{attribute 'linkalways'} 
{attribute 'no_explicit_call' := 'This FB is a CLASS and must be accessed using methods or properties'}
{attribute 'enable_dynamic_creation'}
FUNCTION_BLOCK Node_F_VN_DrawPolygonExp EXTENDS VisionNode
VAR
    ipPoints : _ITcVnContainer;
    ipDestImage : _ITcVnImage;
    aColor : _TcVnVector4_LREAL;
    nThickness : _DINT(1);
    bIsClosed : _BOOL(FALSE);
    eLineType : _ETcVnLineType(ETcVnLineType.TCVN_LT_4_CONNECTED);
    nShift : _UDINT(0);
    hrPrev : _HRESULT(S_OK);
	hresult : _HRESULT(S_OK);
END_VAR

METHOD PUBLIC  Clone : I_Node
VAR
	pNode : POINTER TO Node_F_VN_DrawPolygonExp
;
END_VAR
pNode := __NEW(Node_F_VN_DrawPolygonExp);
Clone := pNode^;
END_METHOD

METHOD FB_init : BOOL
VAR_INPUT
	bInitRetains : BOOL; // if TRUE, the retain variables are initialized (warm start / cold start)
	bInCopyCode : BOOL;  // if TRUE, the instance afterwards gets moved into the copy code (online change)
END_VAR
AddInput('ipPoints', ipPoints);
AddInput('ipDestImage', ipDestImage);
AddInput('aColor', aColor);
AddParameter('nThickness', nThickness);
AddParameter('bIsClosed', bIsClosed);
AddParameter('eLineType', eLineType);
AddParameter('nShift', nShift);
AddInput('hrPrev', hrPrev);
AddOutput('ipDestImage', ipDestImage);
AddOutput('hresult',hresult);
END_METHOD

METHOD PROTECTED OnExecute
hresult.Value := F_VN_DrawPolygonExp(
    ipPoints := ipPoints.Value,
	ipDestImage := ipDestImage.Value,
    aColor := aColor.Value,
    nThickness := nThickness.Value,
    bIsClosed := bIsClosed.Value,
    eLineType := eLineType.Value,
    nShift := nShift.Value,
	hrPrev:= hrPrev.Value);
END_METHOD

METHOD PUBLIC PreExecutionCheck
VAR_INPUT
	Check : I_PreExecutionChecks;
END_VAR
Check.IsTrue(ipPoints.IsValid, 'ipContours must be a valid container');
Check.IsTrue((ipPoints.HasType(TC_GLOBAL_CONST_LIST.ContainerType_Vector_TcVnPoint2_DINT) OR
              ipPoints.HasType(TC_GLOBAL_CONST_LIST.ContainerType_Vector_TcVnPoint2_REAL) OR
              ipPoints.HasType(TC_GLOBAL_CONST_LIST.ContainerType_Vector_TcVnPoint2_LREAL)),
              'ipPoints contains incorrect type');

Check.IsTrue(ipDestImage.IsValid, 'ipDestImage must contain an image');
END_METHOD

END_FUNCTION_BLOCK

(* stored: Version 1.1.0.1, ProductVersion 3.1.4024.15
   POU Node_F_VN_DrawPolygonExp: Id {76832a58-23e2-0b89-399f-7f9b15e7c259}, SpecialFunc None
   Folder Constructor: Id {7ddc0cca-4a75-0c9f-2b9c-a4de12a3c1d3}
   Method Clone: Id {b2564b9b-79e7-00bc-2e7d-c4bf572b6787}
   Method FB_init: Id {96176d5e-4820-01dc-1dbb-f9bfabc9844d}
   Method OnExecute: Id {a6ade25b-ef3d-0de8-1e6f-586831b0cadc}
   Method PreExecutionCheck: Id {531cfd5c-2ac5-03b7-3dcc-0421a5c40439} *)
